// TIA Portal V20 export
FUNCTION "LAL100" : Void   // FC7, FBD
{ S7_Optimized_Access := 'TRUE' }
// stored: SetENOAutomatically false
BEGIN

REGION Network 1: Channel input
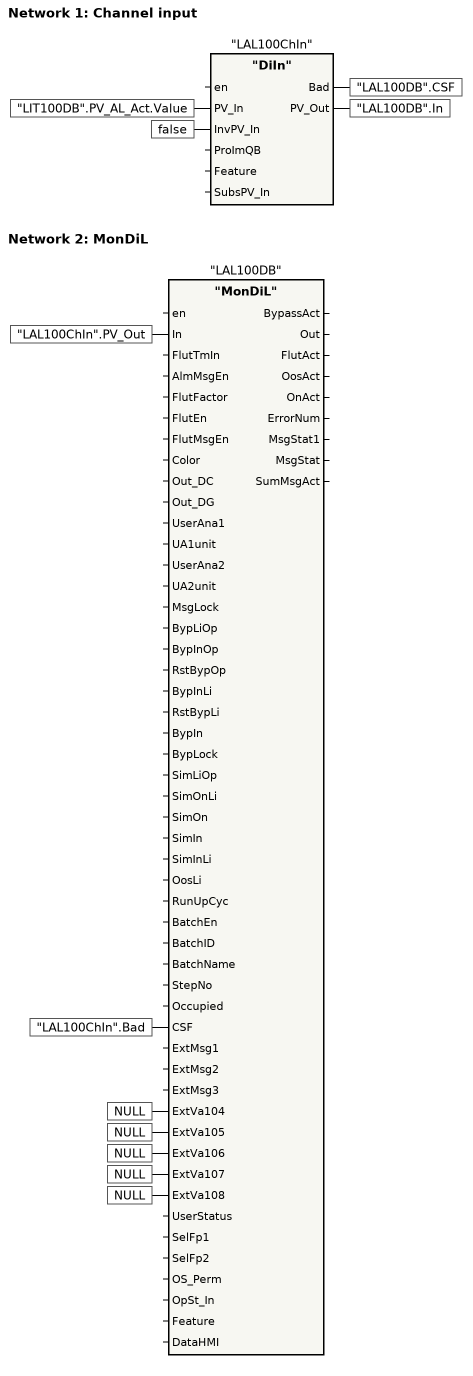
   "LAL100ChIn"(PV_In := "LIT100DB".PV_AL_Act.Value,   // "DiIn"
                InvPV_In := false,
                Bad => "LAL100DB".CSF,
                PV_Out => "LAL100DB".In);
END_REGION

REGION Network 2: MonDiL
   "LAL100DB"(In := "LAL100ChIn".PV_Out,   // "MonDiL"
              CSF := "LAL100ChIn".Bad,
              ExtVa104 := NULL,
              ExtVa105 := NULL,
              ExtVa106 := NULL,
              ExtVa107 := NULL,
              ExtVa108 := NULL);
END_REGION

REGION Network 3: MTP
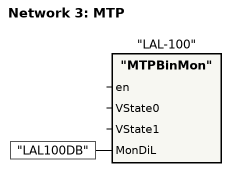
   "LAL-100"(MonDiL := "LAL100DB");   // "MTPBinMon"
END_REGION
END_FUNCTION
